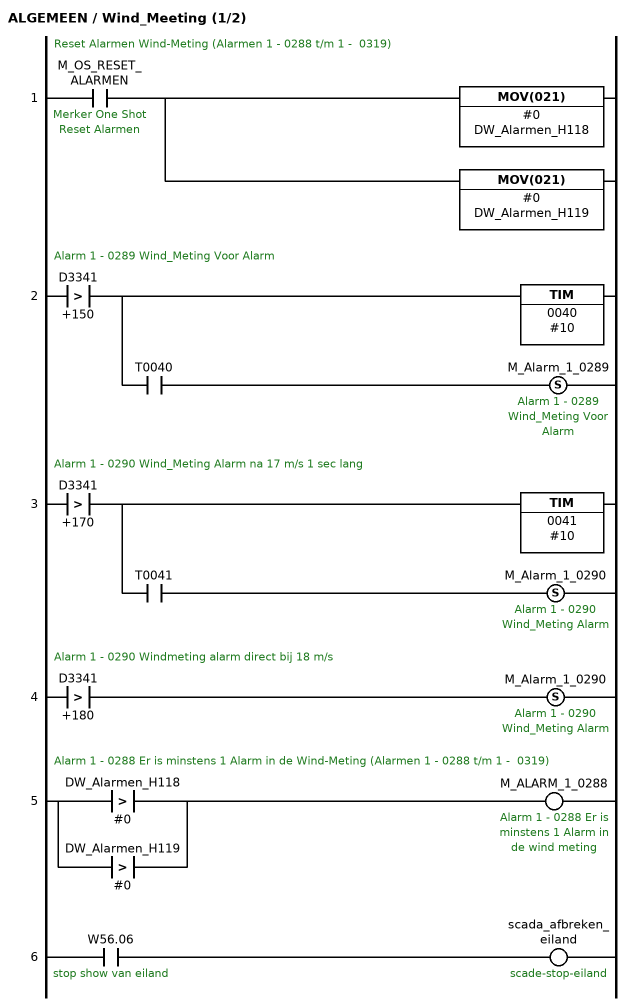
; [picture p72: ALGEMEEN / Wind_Meeting, rungs 1-6]
; rung 1: Reset Alarmen Wind-Meting (Alarmen 1 - 0288 t/m 1 -  0319)
LD M_OS_RESET_ALARMEN  ; Merker One Shot Reset Alarmen
MOV(021) #0 DW_Alarmen_H118
MOV(021) #0 DW_Alarmen_H119
; rung 2: Alarm 1 - 0289 Wind_Meting Voor Alarm
LD>S(322) D3341 +150
TIM 0040 #10
AND T0040
SET M_Alarm_1_0289  ; Alarm 1 - 0289 Wind_Meting Voor Alarm
; rung 3: Alarm 1 - 0290 Wind_Meting Alarm na 17 m/s 1 sec lang
LD>S(322) D3341 +170
TIM 0041 #10
AND T0041
SET M_Alarm_1_0290  ; Alarm 1 - 0290 Wind_Meting Alarm
; rung 4: Alarm 1 - 0290 Windmeting alarm direct bij 18 m/s
LD>S(322) D3341 +180
SET M_Alarm_1_0290  ; Alarm 1 - 0290 Wind_Meting Alarm
; rung 5: Alarm 1 - 0288 Er is minstens 1 Alarm in de Wind-Meting (Alarmen 1 - 0288 t/m 1 -  0319)
LD>(320) DW_Alarmen_H118 #0
OR>(320) DW_Alarmen_H119 #0
OUT M_ALARM_1_0288  ; Alarm 1 - 0288 Er is minstens 1 Alarm in de wind meting
; rung 6
LD W56.06  ; stop show van eiland
OUT scada_afbreken_eiland  ; scade-stop-eiland

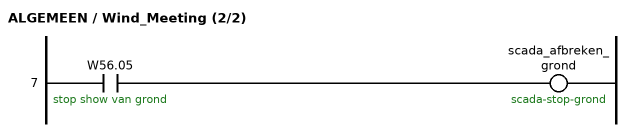
; rung 7
LD W56.05  ; stop show van grond
OUT scada_afbreken_grond  ; scada-stop-grond

### Section Alarm_Handler

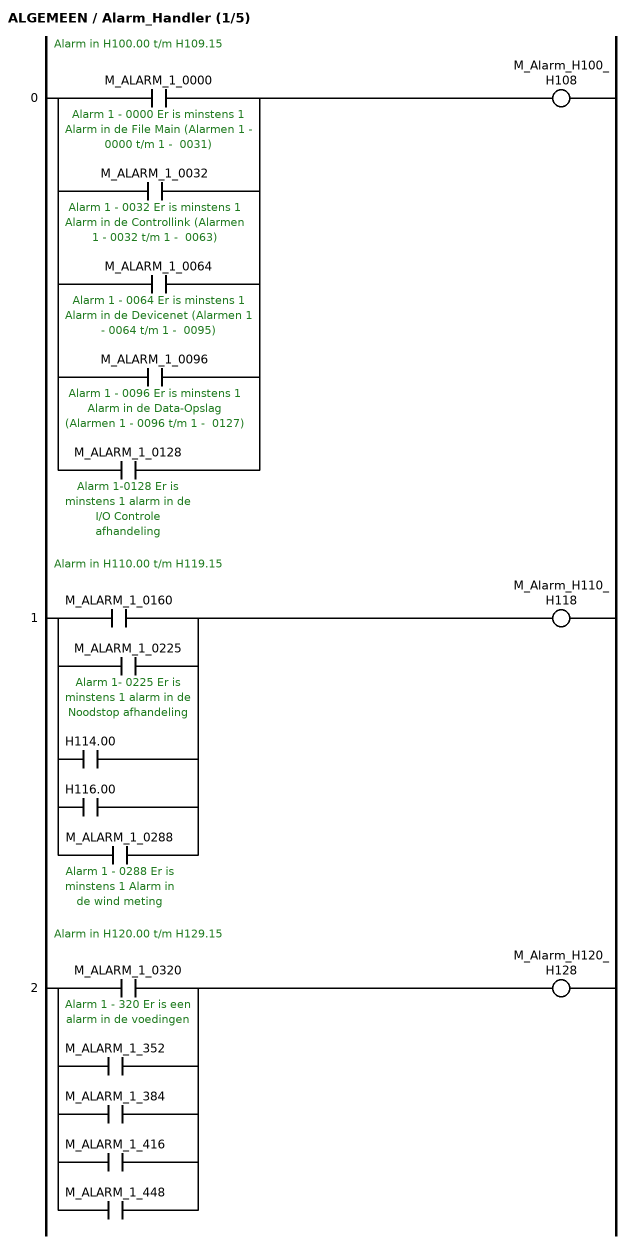
; rung 0: Alarm in H100.00 t/m H109.15
LD M_ALARM_1_0000  ; Alarm 1 - 0000 Er is minstens 1 Alarm in de File Main (Alarmen 1 - 0000 t/m 1 -  0031)
OR M_ALARM_1_0032  ; Alarm 1 - 0032 Er is minstens 1 Alarm in de Controllink (Alarmen 1 - 0032 t/m 1 -  0063)
OR M_ALARM_1_0064  ; Alarm 1 - 0064 Er is minstens 1 Alarm in de Devicenet (Alarmen 1 - 0064 t/m 1 -  0095)
OR M_ALARM_1_0096  ; Alarm 1 - 0096 Er is minstens 1 Alarm in de Data-Opslag (Alarmen 1 - 0096 t/m 1 -  0127)
OR M_ALARM_1_0128  ; Alarm 1-0128 Er is minstens 1 alarm in de I/O Controle afhandeling
OUT M_Alarm_H100_H108
; rung 1: Alarm in H110.00 t/m H119.15
LD M_ALARM_1_0160
OR M_ALARM_1_0225  ; Alarm 1- 0225 Er is minstens 1 alarm in de Noodstop afhandeling
OR H114.00
OR H116.00
OR M_ALARM_1_0288  ; Alarm 1 - 0288 Er is minstens 1 Alarm in de wind meting
OUT M_Alarm_H110_H118
; rung 2: Alarm in H120.00 t/m H129.15
LD M_ALARM_1_0320  ; Alarm 1 - 320 Er is een alarm in de voedingen
OR M_ALARM_1_352
OR M_ALARM_1_384
OR M_ALARM_1_416
OR M_ALARM_1_448
OUT M_Alarm_H120_H128

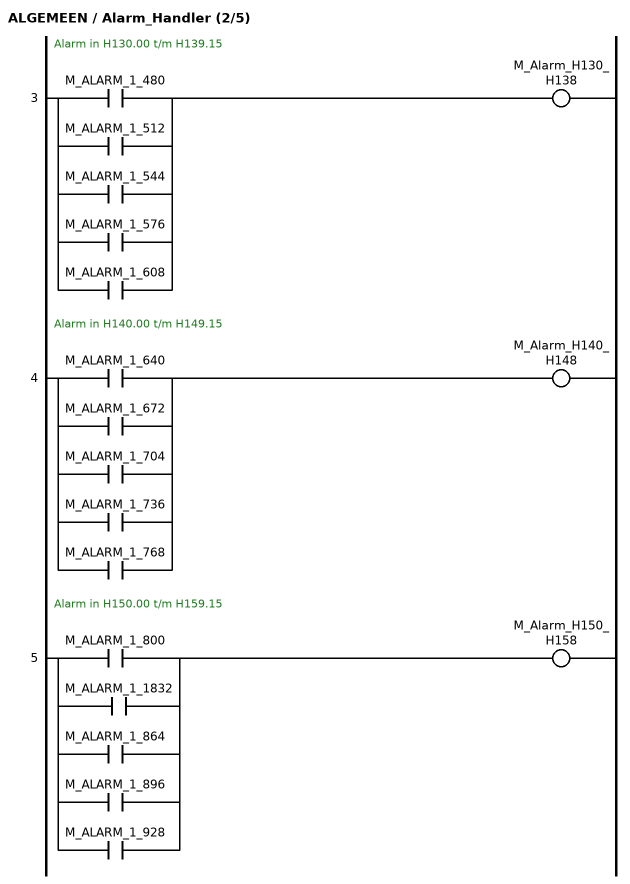
; rung 3: Alarm in H130.00 t/m H139.15
LD M_ALARM_1_480
OR M_ALARM_1_512
OR M_ALARM_1_544
OR M_ALARM_1_576
OR M_ALARM_1_608
OUT M_Alarm_H130_H138
; rung 4: Alarm in H140.00 t/m H149.15
LD M_ALARM_1_640
OR M_ALARM_1_672
OR M_ALARM_1_704
OR M_ALARM_1_736
OR M_ALARM_1_768
OUT M_Alarm_H140_H148
; rung 5: Alarm in H150.00 t/m H159.15
LD M_ALARM_1_800
OR M_ALARM_1_1832
OR M_ALARM_1_864
OR M_ALARM_1_896
OR M_ALARM_1_928
OUT M_Alarm_H150_H158

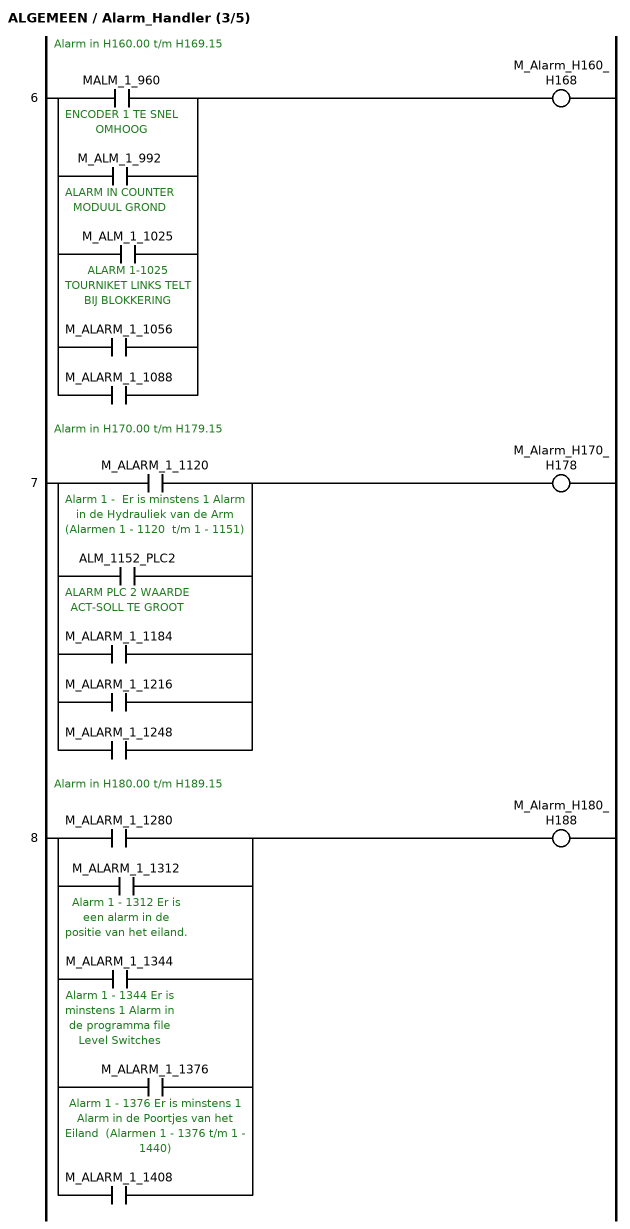
; rung 6: Alarm in H160.00 t/m H169.15
LD MALM_1_960  ; ENCODER 1 TE SNEL OMHOOG
OR M_ALM_1_992  ; ALARM IN COUNTER MODUUL GROND
OR M_ALM_1_1025  ; ALARM 1-1025 TOURNIKET LINKS TELT BIJ BLOKKERING
OR M_ALARM_1_1056
OR M_ALARM_1_1088
OUT M_Alarm_H160_H168
; rung 7: Alarm in H170.00 t/m H179.15
LD M_ALARM_1_1120  ; Alarm 1 -  Er is minstens 1 Alarm in de Hydrauliek van de Arm  (Alarmen 1 - 1120  t/m 1 - 1151)
OR ALM_1152_PLC2  ; ALARM PLC 2 WAARDE ACT-SOLL TE GROOT
OR M_ALARM_1_1184
OR M_ALARM_1_1216
OR M_ALARM_1_1248
OUT M_Alarm_H170_H178
; rung 8: Alarm in H180.00 t/m H189.15
LD M_ALARM_1_1280
OR M_ALARM_1_1312  ; Alarm 1 - 1312 Er is een alarm in de positie van het eiland.
OR M_ALARM_1_1344  ; Alarm 1 - 1344 Er is minstens 1 Alarm in de programma file Level Switches
OR M_ALARM_1_1376  ; Alarm 1 - 1376 Er is minstens 1 Alarm in de Poortjes van het Eiland  (Alarmen 1 - 1376 t/m 1 - 1440)
OR M_ALARM_1_1408
OUT M_Alarm_H180_H188

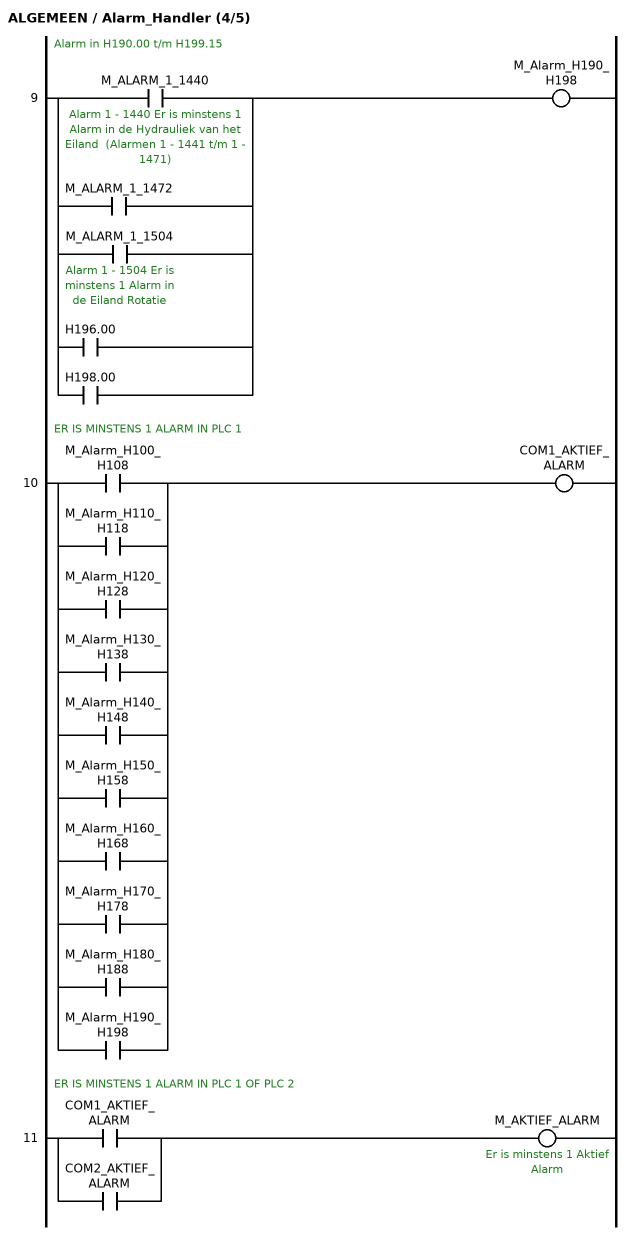
; rung 9: Alarm in H190.00 t/m H199.15
LD M_ALARM_1_1440  ; Alarm 1 - 1440 Er is minstens 1 Alarm in de Hydrauliek van het Eiland  (Alarmen 1 - 1441 t/m 1 - 1471)
OR M_ALARM_1_1472
OR M_ALARM_1_1504  ; Alarm 1 - 1504 Er is minstens 1 Alarm in de Eiland Rotatie
OR H196.00
OR H198.00
OUT M_Alarm_H190_H198
; rung 10: ER IS MINSTENS 1 ALARM IN PLC 1
LD M_Alarm_H100_H108
OR M_Alarm_H110_H118
OR M_Alarm_H120_H128
OR M_Alarm_H130_H138
OR M_Alarm_H140_H148
OR M_Alarm_H150_H158
OR M_Alarm_H160_H168
OR M_Alarm_H170_H178
OR M_Alarm_H180_H188
OR M_Alarm_H190_H198
OUT COM1_AKTIEF_ALARM
; rung 11: ER IS MINSTENS 1 ALARM IN PLC 1 OF PLC 2
LD COM1_AKTIEF_ALARM
OR COM2_AKTIEF_ALARM
OUT M_AKTIEF_ALARM  ; Er is minstens 1 Aktief Alarm

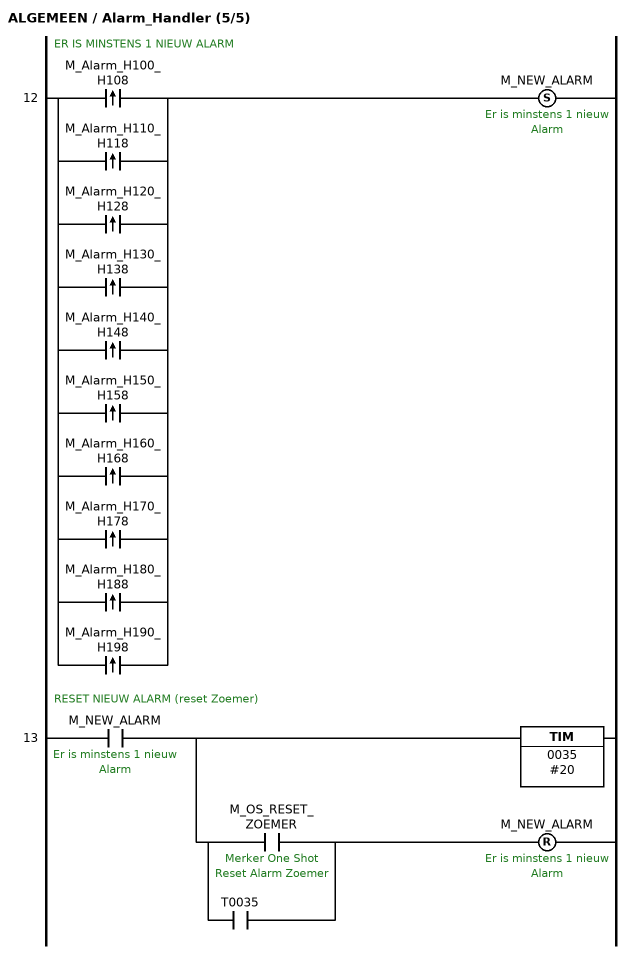
; rung 12: ER IS MINSTENS 1 NIEUW ALARM
@LD M_Alarm_H100_H108
@OR M_Alarm_H110_H118
@OR M_Alarm_H120_H128
@OR M_Alarm_H130_H138
@OR M_Alarm_H140_H148
@OR M_Alarm_H150_H158
@OR M_Alarm_H160_H168
@OR M_Alarm_H170_H178
@OR M_Alarm_H180_H188
@OR M_Alarm_H190_H198
SET M_NEW_ALARM  ; Er is minstens 1 nieuw Alarm
; rung 13: RESET NIEUW ALARM (reset Zoemer)
LD M_NEW_ALARM  ; Er is minstens 1 nieuw Alarm
TIM 0035 #20
LD M_OS_RESET_ZOEMER  ; Merker One Shot Reset Alarm Zoemer
OR T0035
ANDLD
RSET M_NEW_ALARM  ; Er is minstens 1 nieuw Alarm

### Section Einde_Algemeen
; rung 0
END(001)

## Program BEDIENING_SIGNAAL (cyclic task 1)
Local symbols
M_Hydrauliek_x_tijd_aan W56.03 BOOL  ; Hydrauliek x tijd laten door lopen nadat mode is veranderd

### Section Bediening_Scada

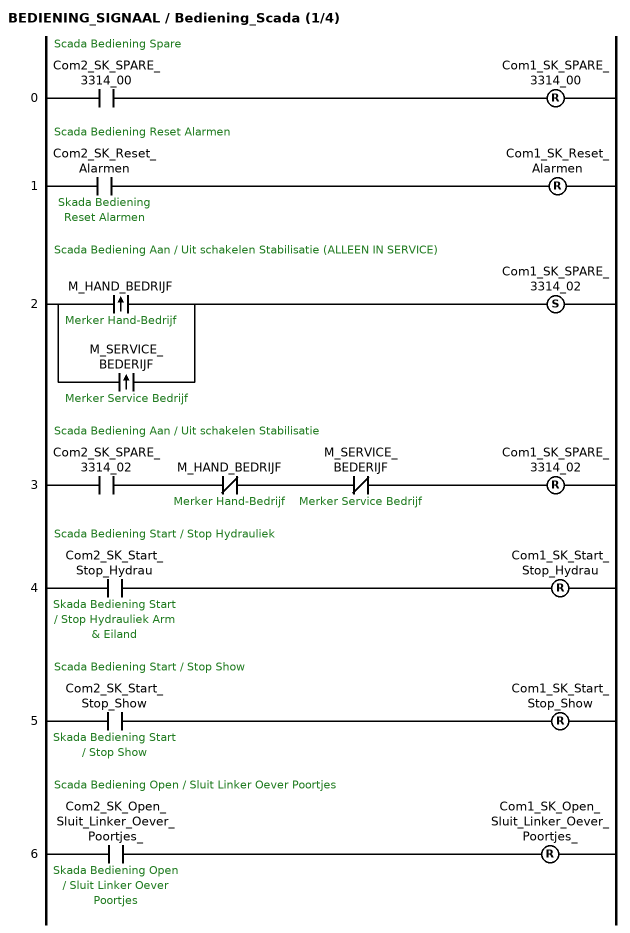
; rung 0: Scada Bediening Spare
LD Com2_SK_SPARE_3314_00
RSET Com1_SK_SPARE_3314_00
; rung 1: Scada Bediening Reset Alarmen
LD Com2_SK_Reset_Alarmen  ; Skada Bediening Reset Alarmen
RSET Com1_SK_Reset_Alarmen
; rung 2: Scada Bediening Aan / Uit schakelen Stabilisatie (ALLEEN IN SERVICE)
@LD M_HAND_BEDRIJF  ; Merker Hand-Bedrijf
@OR M_SERVICE_BEDERIJF  ; Merker Service Bedrijf
SET Com1_SK_SPARE_3314_02
; rung 3: Scada Bediening Aan / Uit schakelen Stabilisatie
LD Com2_SK_SPARE_3314_02
ANDNOT M_HAND_BEDRIJF  ; Merker Hand-Bedrijf
ANDNOT M_SERVICE_BEDERIJF  ; Merker Service Bedrijf
RSET Com1_SK_SPARE_3314_02
; rung 4: Scada Bediening Start / Stop Hydrauliek
LD Com2_SK_Start_Stop_Hydrau  ; Skada Bediening Start / Stop Hydrauliek Arm & Eiland
RSET Com1_SK_Start_Stop_Hydrau
; rung 5: Scada Bediening Start / Stop Show
LD Com2_SK_Start_Stop_Show  ; Skada Bediening Start / Stop Show
RSET Com1_SK_Start_Stop_Show
; rung 6: Scada Bediening Open / Sluit Linker Oever Poortjes
LD Com2_SK_Open_Sluit_Linker_Oever_Poortjes_  ; Skada Bediening Open / Sluit Linker Oever Poortjes
RSET Com1_SK_Open_Sluit_Linker_Oever_Poortjes_

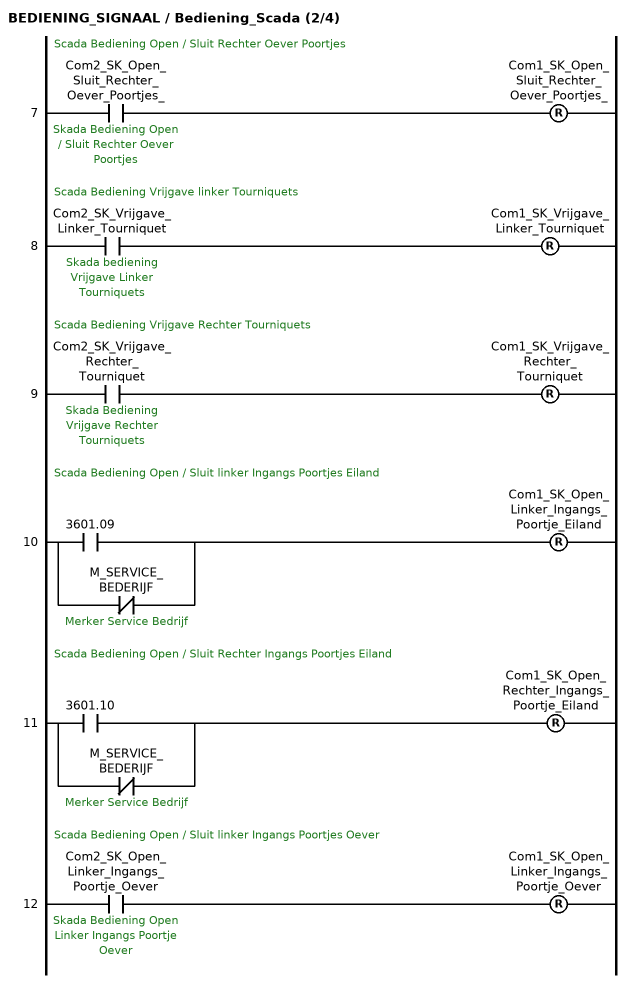
; rung 7: Scada Bediening Open / Sluit Rechter Oever Poortjes
LD Com2_SK_Open_Sluit_Rechter_Oever_Poortjes_  ; Skada Bediening Open / Sluit Rechter Oever Poortjes
RSET Com1_SK_Open_Sluit_Rechter_Oever_Poortjes_
; rung 8: Scada Bediening Vrijgave linker Tourniquets
LD Com2_SK_Vrijgave_Linker_Tourniquet  ; Skada bediening Vrijgave Linker Tourniquets
RSET Com1_SK_Vrijgave_Linker_Tourniquet
; rung 9: Scada Bediening Vrijgave Rechter Tourniquets
LD Com2_SK_Vrijgave_Rechter_Tourniquet  ; Skada Bediening Vrijgave Rechter Tourniquets
RSET Com1_SK_Vrijgave_Rechter_Tourniquet
; rung 10: Scada Bediening Open / Sluit linker Ingangs Poortjes Eiland
LD 3601.09
ORNOT M_SERVICE_BEDERIJF  ; Merker Service Bedrijf
RSET Com1_SK_Open_Linker_Ingangs_Poortje_Eiland
; rung 11: Scada Bediening Open / Sluit Rechter Ingangs Poortjes Eiland
LD 3601.10
ORNOT M_SERVICE_BEDERIJF  ; Merker Service Bedrijf
RSET Com1_SK_Open_Rechter_Ingangs_Poortje_Eiland
; rung 12: Scada Bediening Open / Sluit linker Ingangs Poortjes Oever
LD Com2_SK_Open_Linker_Ingangs_Poortje_Oever  ; Skada Bediening Open Linker Ingangs Poortje Oever
RSET Com1_SK_Open_Linker_Ingangs_Poortje_Oever

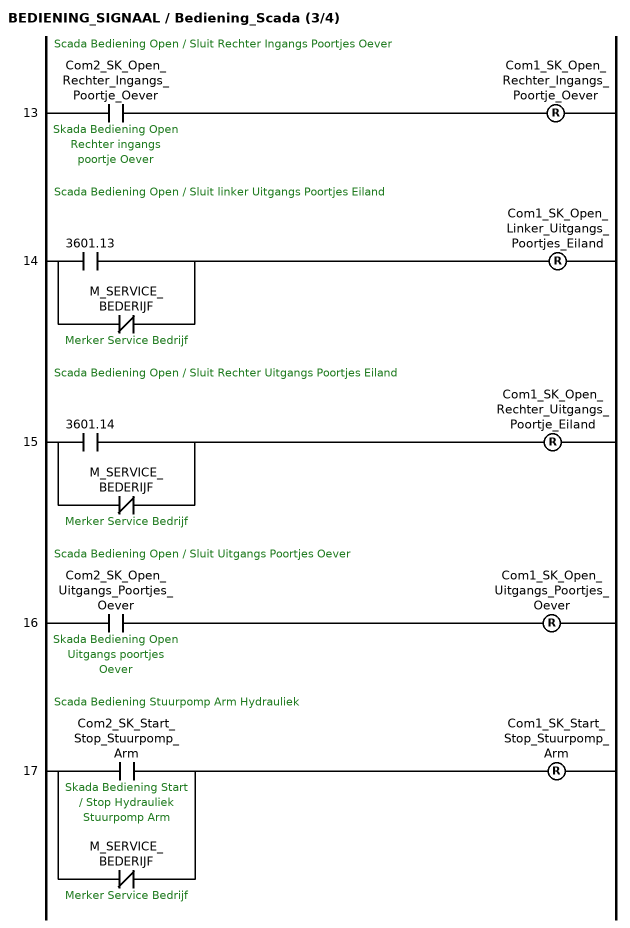
; rung 13: Scada Bediening Open / Sluit Rechter Ingangs Poortjes Oever
LD Com2_SK_Open_Rechter_Ingangs_Poortje_Oever  ; Skada Bediening Open Rechter ingangs poortje Oever
RSET Com1_SK_Open_Rechter_Ingangs_Poortje_Oever
; rung 14: Scada Bediening Open / Sluit linker Uitgangs Poortjes Eiland
LD 3601.13
ORNOT M_SERVICE_BEDERIJF  ; Merker Service Bedrijf
RSET Com1_SK_Open_Linker_Uitgangs_Poortjes_Eiland
; rung 15: Scada Bediening Open / Sluit Rechter Uitgangs Poortjes Eiland
LD 3601.14
ORNOT M_SERVICE_BEDERIJF  ; Merker Service Bedrijf
RSET Com1_SK_Open_Rechter_Uitgangs_Poortje_Eiland
; rung 16: Scada Bediening Open / Sluit Uitgangs Poortjes Oever
LD Com2_SK_Open_Uitgangs_Poortjes_Oever  ; Skada Bediening Open Uitgangs poortjes Oever
RSET Com1_SK_Open_Uitgangs_Poortjes_Oever
; rung 17: Scada Bediening Stuurpomp Arm Hydrauliek
LD Com2_SK_Start_Stop_Stuurpomp_Arm  ; Skada Bediening Start / Stop Hydrauliek Stuurpomp Arm
ORNOT M_SERVICE_BEDERIJF  ; Merker Service Bedrijf
RSET Com1_SK_Start_Stop_Stuurpomp_Arm

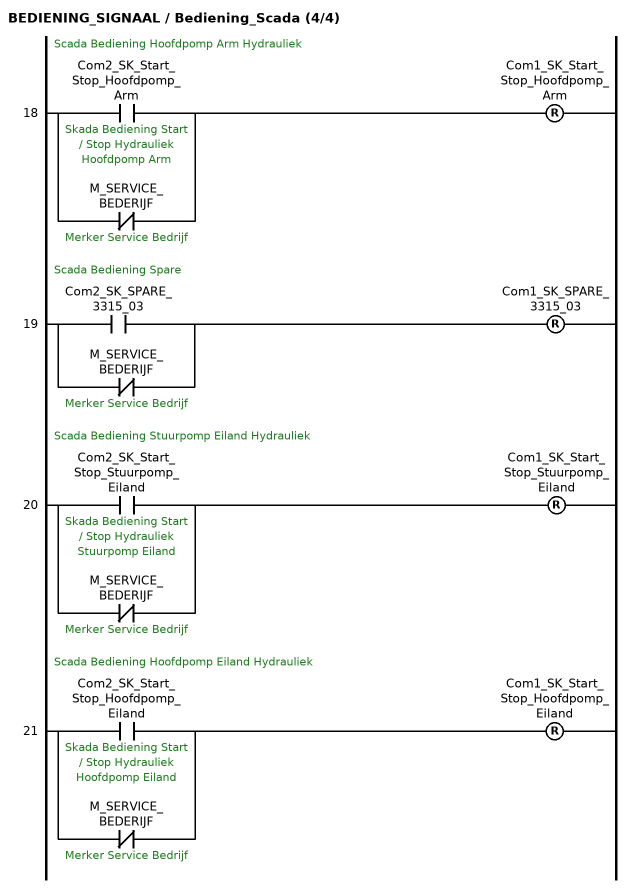
; rung 18: Scada Bediening Hoofdpomp Arm Hydrauliek
LD Com2_SK_Start_Stop_Hoofdpomp_Arm  ; Skada Bediening Start / Stop Hydrauliek Hoofdpomp Arm
ORNOT M_SERVICE_BEDERIJF  ; Merker Service Bedrijf
RSET Com1_SK_Start_Stop_Hoofdpomp_Arm
; rung 19: Scada Bediening Spare
LD Com2_SK_SPARE_3315_03
ORNOT M_SERVICE_BEDERIJF  ; Merker Service Bedrijf
RSET Com1_SK_SPARE_3315_03
; rung 20: Scada Bediening Stuurpomp Eiland Hydrauliek
LD Com2_SK_Start_Stop_Stuurpomp_Eiland  ; Skada Bediening Start / Stop Hydrauliek Stuurpomp Eiland
ORNOT M_SERVICE_BEDERIJF  ; Merker Service Bedrijf
RSET Com1_SK_Start_Stop_Stuurpomp_Eiland
; rung 21: Scada Bediening Hoofdpomp Eiland Hydrauliek
LD Com2_SK_Start_Stop_Hoofdpomp_Eiland  ; Skada Bediening Start / Stop Hydrauliek Hoofdpomp Eiland
ORNOT M_SERVICE_BEDERIJF  ; Merker Service Bedrijf
RSET Com1_SK_Start_Stop_Hoofdpomp_Eiland

### Section Signalering_Scada

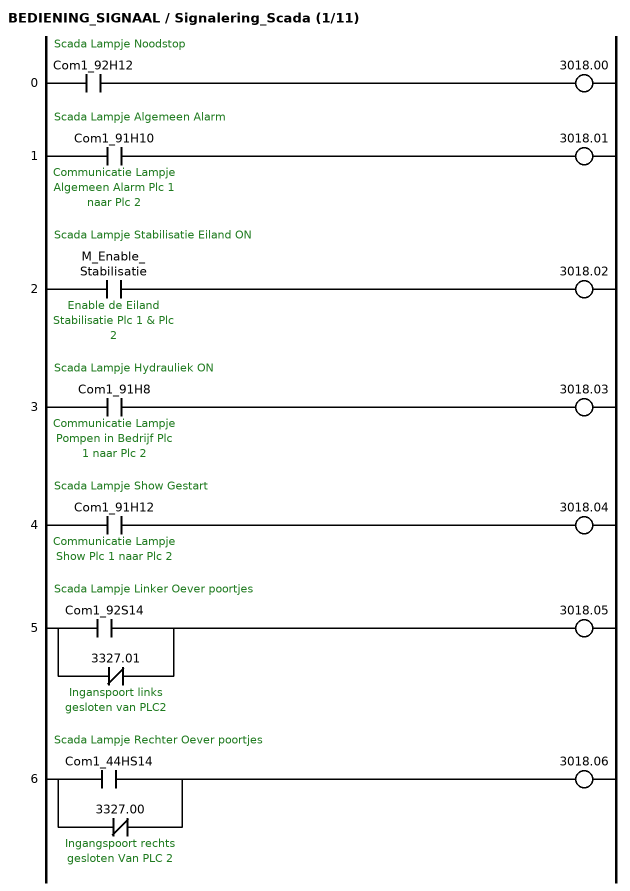
; rung 0: Scada Lampje Noodstop
LD Com1_92H12
OUT 3018.00
; rung 1: Scada Lampje Algemeen Alarm
LD Com1_91H10  ; Communicatie Lampje Algemeen Alarm Plc 1 naar Plc 2
OUT 3018.01
; rung 2: Scada Lampje Stabilisatie Eiland ON
LD M_Enable_Stabilisatie  ; Enable de Eiland Stabilisatie Plc 1 & Plc 2
OUT 3018.02
; rung 3: Scada Lampje Hydrauliek ON
LD Com1_91H8  ; Communicatie Lampje Pompen in Bedrijf Plc 1 naar Plc 2
OUT 3018.03
; rung 4: Scada Lampje Show Gestart
LD Com1_91H12  ; Communicatie Lampje Show Plc 1 naar Plc 2
OUT 3018.04
; rung 5: Scada Lampje Linker Oever poortjes
LD Com1_92S14
ORNOT 3327.01  ; Inganspoort links gesloten van PLC2
OUT 3018.05
; rung 6: Scada Lampje Rechter Oever poortjes
LD Com1_44HS14
ORNOT 3327.00  ; Ingangspoort rechts gesloten Van PLC 2
OUT 3018.06

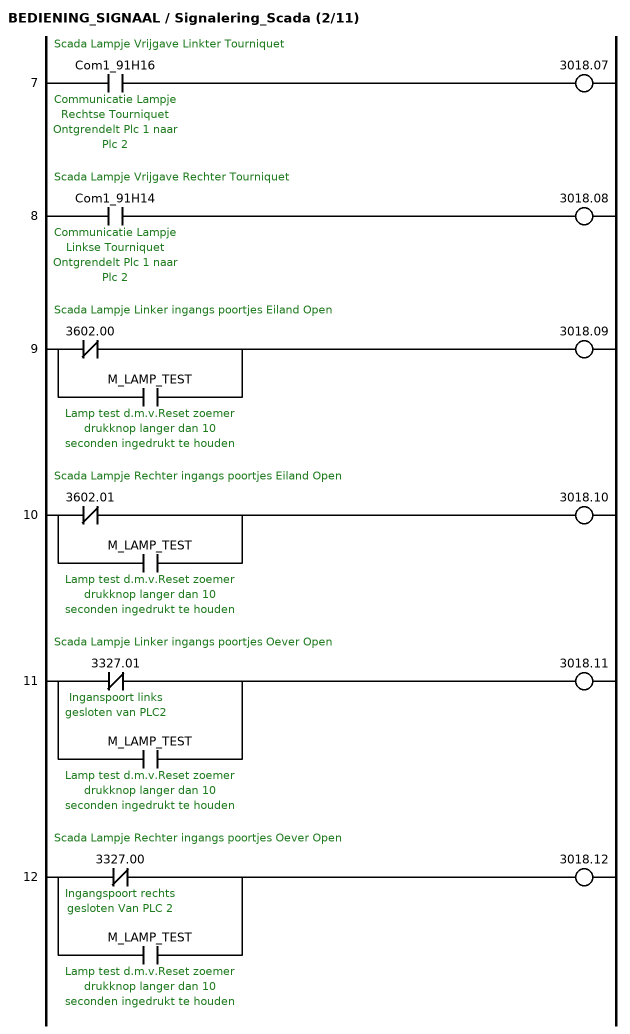
; rung 7: Scada Lampje Vrijgave Linkter Tourniquet
LD Com1_91H16  ; Communicatie Lampje Rechtse Tourniquet Ontgrendelt Plc 1 naar Plc 2
OUT 3018.07
; rung 8: Scada Lampje Vrijgave Rechter Tourniquet
LD Com1_91H14  ; Communicatie Lampje Linkse Tourniquet Ontgrendelt Plc 1 naar Plc 2
OUT 3018.08
; rung 9: Scada Lampje Linker ingangs poortjes Eiland Open
LDNOT 3602.00
OR M_LAMP_TEST  ; Lamp test d.m.v.Reset zoemer drukknop langer dan 10 seconden ingedrukt te houden
OUT 3018.09
; rung 10: Scada Lampje Rechter ingangs poortjes Eiland Open
LDNOT 3602.01
OR M_LAMP_TEST  ; Lamp test d.m.v.Reset zoemer drukknop langer dan 10 seconden ingedrukt te houden
OUT 3018.10
; rung 11: Scada Lampje Linker ingangs poortjes Oever Open
LDNOT 3327.01  ; Inganspoort links gesloten van PLC2
OR M_LAMP_TEST  ; Lamp test d.m.v.Reset zoemer drukknop langer dan 10 seconden ingedrukt te houden
OUT 3018.11
; rung 12: Scada Lampje Rechter ingangs poortjes Oever Open
LDNOT 3327.00  ; Ingangspoort rechts gesloten Van PLC 2
OR M_LAMP_TEST  ; Lamp test d.m.v.Reset zoemer drukknop langer dan 10 seconden ingedrukt te houden
OUT 3018.12

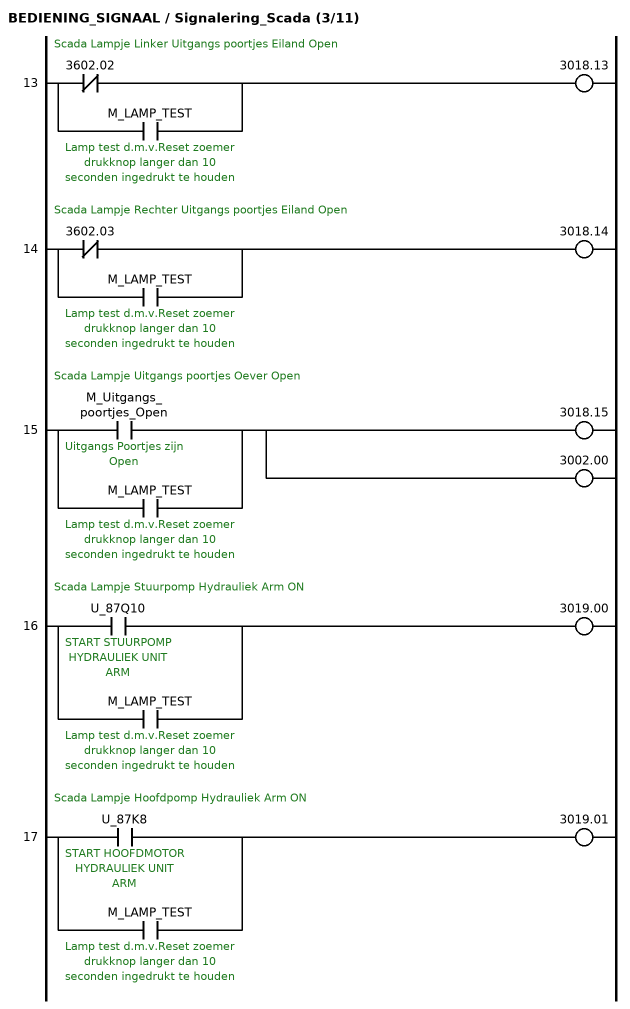
; rung 13: Scada Lampje Linker Uitgangs poortjes Eiland Open
LDNOT 3602.02
OR M_LAMP_TEST  ; Lamp test d.m.v.Reset zoemer drukknop langer dan 10 seconden ingedrukt te houden
OUT 3018.13
; rung 14: Scada Lampje Rechter Uitgangs poortjes Eiland Open
LDNOT 3602.03
OR M_LAMP_TEST  ; Lamp test d.m.v.Reset zoemer drukknop langer dan 10 seconden ingedrukt te houden
OUT 3018.14
; rung 15: Scada Lampje Uitgangs poortjes Oever Open
LD M_Uitgangs_poortjes_Open  ; Uitgangs Poortjes zijn Open
OR M_LAMP_TEST  ; Lamp test d.m.v.Reset zoemer drukknop langer dan 10 seconden ingedrukt te houden
OUT 3018.15
OUT 3002.00
; rung 16: Scada Lampje Stuurpomp Hydrauliek Arm ON
LD U_87Q10  ; START STUURPOMP HYDRAULIEK UNIT ARM
OR M_LAMP_TEST  ; Lamp test d.m.v.Reset zoemer drukknop langer dan 10 seconden ingedrukt te houden
OUT 3019.00
; rung 17: Scada Lampje Hoofdpomp Hydrauliek Arm ON
LD U_87K8  ; START HOOFDMOTOR HYDRAULIEK UNIT ARM
OR M_LAMP_TEST  ; Lamp test d.m.v.Reset zoemer drukknop langer dan 10 seconden ingedrukt te houden
OUT 3019.01

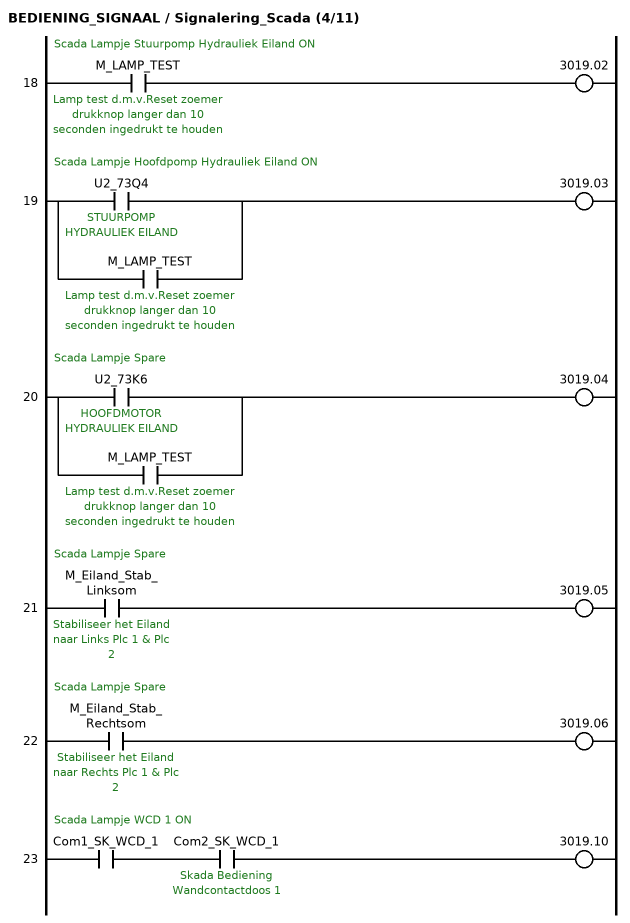
; rung 18: Scada Lampje Stuurpomp Hydrauliek Eiland ON
LD M_LAMP_TEST  ; Lamp test d.m.v.Reset zoemer drukknop langer dan 10 seconden ingedrukt te houden
OUT 3019.02
; rung 19: Scada Lampje Hoofdpomp Hydrauliek Eiland ON
LD U2_73Q4  ; STUURPOMP HYDRAULIEK EILAND
OR M_LAMP_TEST  ; Lamp test d.m.v.Reset zoemer drukknop langer dan 10 seconden ingedrukt te houden
OUT 3019.03
; rung 20: Scada Lampje Spare
LD U2_73K6  ; HOOFDMOTOR HYDRAULIEK EILAND
OR M_LAMP_TEST  ; Lamp test d.m.v.Reset zoemer drukknop langer dan 10 seconden ingedrukt te houden
OUT 3019.04
; rung 21: Scada Lampje Spare
LD M_Eiland_Stab_Linksom  ; Stabiliseer het Eiland naar Links Plc 1 & Plc 2
OUT 3019.05
; rung 22: Scada Lampje Spare
LD M_Eiland_Stab_Rechtsom  ; Stabiliseer het Eiland naar Rechts Plc 1 & Plc 2
OUT 3019.06
; rung 23: Scada Lampje WCD 1 ON
LD Com1_SK_WCD_1
AND Com2_SK_WCD_1  ; Skada Bediening Wandcontactdoos 1
OUT 3019.10

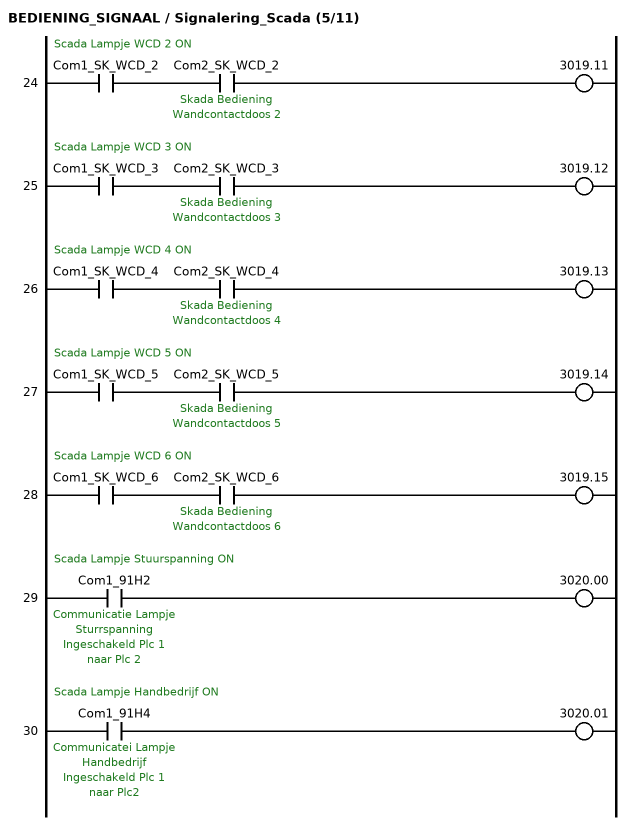
; rung 24: Scada Lampje WCD 2 ON
LD Com1_SK_WCD_2
AND Com2_SK_WCD_2  ; Skada Bediening Wandcontactdoos 2
OUT 3019.11
; rung 25: Scada Lampje WCD 3 ON
LD Com1_SK_WCD_3
AND Com2_SK_WCD_3  ; Skada Bediening Wandcontactdoos 3
OUT 3019.12
; rung 26: Scada Lampje WCD 4 ON
LD Com1_SK_WCD_4
AND Com2_SK_WCD_4  ; Skada Bediening Wandcontactdoos 4
OUT 3019.13
; rung 27: Scada Lampje WCD 5 ON
LD Com1_SK_WCD_5
AND Com2_SK_WCD_5  ; Skada Bediening Wandcontactdoos 5
OUT 3019.14
; rung 28: Scada Lampje WCD 6 ON
LD Com1_SK_WCD_6
AND Com2_SK_WCD_6  ; Skada Bediening Wandcontactdoos 6
OUT 3019.15
; rung 29: Scada Lampje Stuurspanning ON
LD Com1_91H2  ; Communicatie Lampje Sturrspanning Ingeschakeld Plc 1 naar Plc 2
OUT 3020.00
; rung 30: Scada Lampje Handbedrijf ON
LD Com1_91H4  ; Communicatei Lampje Handbedrijf Ingeschakeld Plc 1 naar Plc2
OUT 3020.01

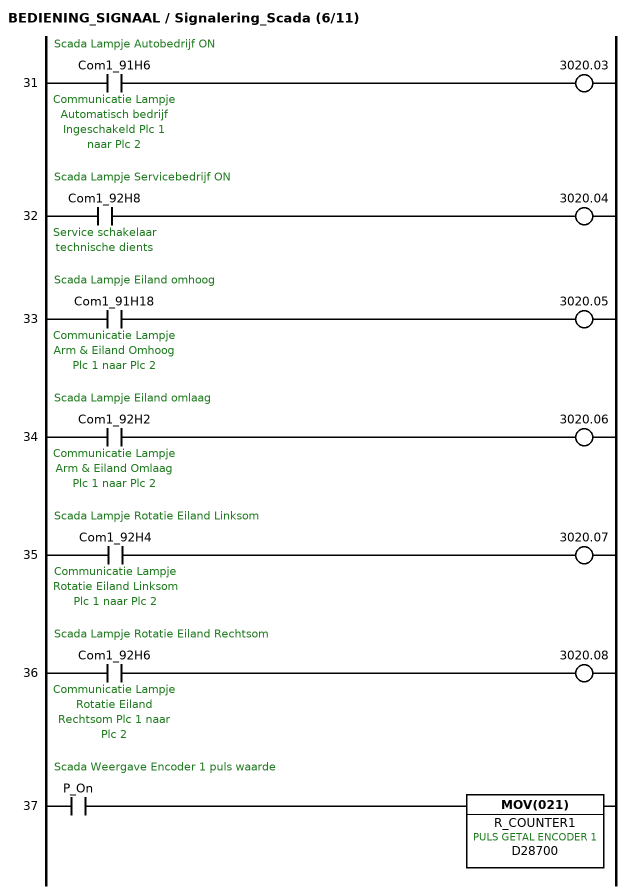
; rung 31: Scada Lampje Autobedrijf ON
LD Com1_91H6  ; Communicatie Lampje Automatisch bedrijf Ingeschakeld Plc 1 naar Plc 2
OUT 3020.03
; rung 32: Scada Lampje Servicebedrijf ON
LD Com1_92H8  ; Service schakelaar technische dients
OUT 3020.04
; rung 33: Scada Lampje Eiland omhoog
LD Com1_91H18  ; Communicatie Lampje Arm & Eiland Omhoog Plc 1 naar Plc 2
OUT 3020.05
; rung 34: Scada Lampje Eiland omlaag
LD Com1_92H2  ; Communicatie Lampje Arm & Eiland Omlaag Plc 1 naar Plc 2
OUT 3020.06
; rung 35: Scada Lampje Rotatie Eiland Linksom
LD Com1_92H4  ; Communicatie Lampje Rotatie Eiland Linksom Plc 1 naar Plc 2
OUT 3020.07
; rung 36: Scada Lampje Rotatie Eiland Rechtsom
LD Com1_92H6  ; Communicatie Lampje Rotatie Eiland Rechtsom Plc 1 naar Plc 2
OUT 3020.08
; rung 37: Scada Weergave Encoder 1 puls waarde
LD P_On
MOV(021) R_COUNTER1 D28700  ; PULS GETAL ENCODER 1

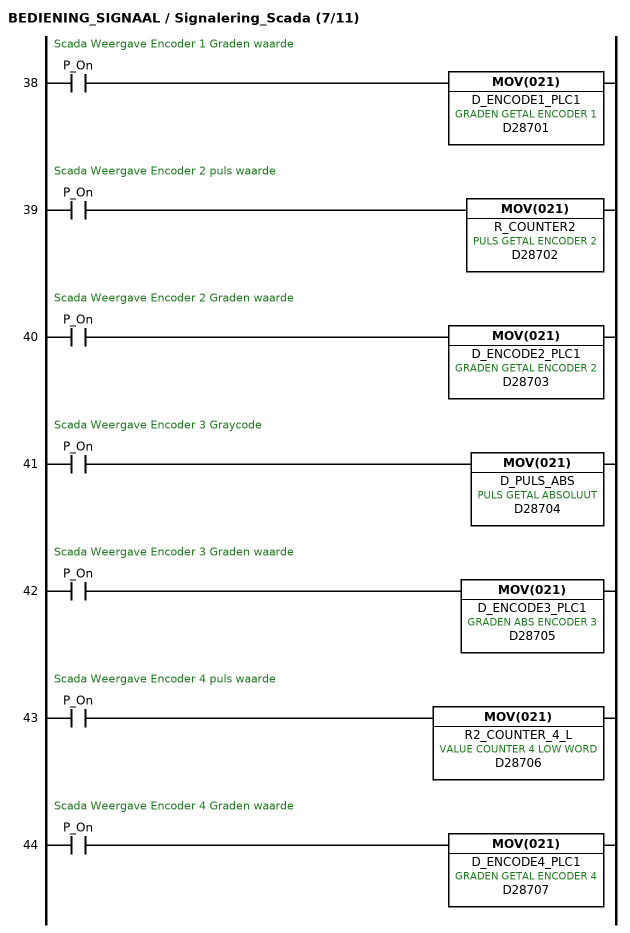
; rung 38: Scada Weergave Encoder 1 Graden waarde
LD P_On
MOV(021) D_ENCODE1_PLC1 D28701  ; GRADEN GETAL ENCODER 1
; rung 39: Scada Weergave Encoder 2 puls waarde
LD P_On
MOV(021) R_COUNTER2 D28702  ; PULS GETAL ENCODER 2
; rung 40: Scada Weergave Encoder 2 Graden waarde
LD P_On
MOV(021) D_ENCODE2_PLC1 D28703  ; GRADEN GETAL ENCODER 2
; rung 41: Scada Weergave Encoder 3 Graycode
LD P_On
MOV(021) D_PULS_ABS D28704  ; PULS GETAL ABSOLUUT
; rung 42: Scada Weergave Encoder 3 Graden waarde
LD P_On
MOV(021) D_ENCODE3_PLC1 D28705  ; GRADEN ABS ENCODER 3
; rung 43: Scada Weergave Encoder 4 puls waarde
LD P_On
MOV(021) R2_COUNTER_4_L D28706  ; VALUE COUNTER 4 LOW WORD
; rung 44: Scada Weergave Encoder 4 Graden waarde
LD P_On
MOV(021) D_ENCODE4_PLC1 D28707  ; GRADEN GETAL ENCODER 4

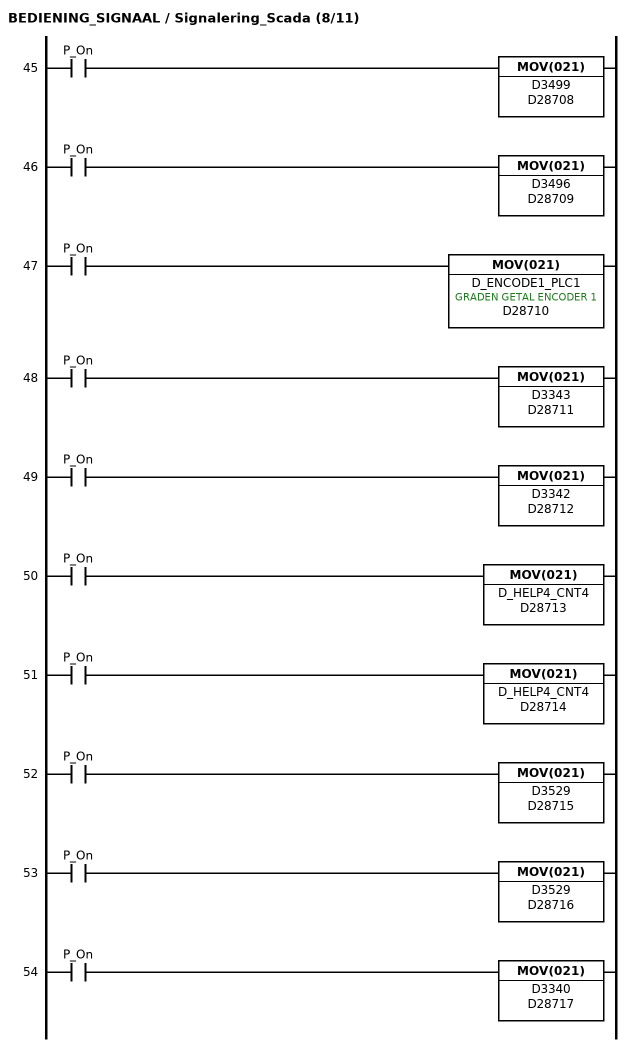
; rung 45
LD P_On
MOV(021) D3499 D28708
; rung 46
LD P_On
MOV(021) D3496 D28709
; rung 47
LD P_On
MOV(021) D_ENCODE1_PLC1 D28710  ; GRADEN GETAL ENCODER 1
; rung 48
LD P_On
MOV(021) D3343 D28711
; rung 49
LD P_On
MOV(021) D3342 D28712
; rung 50
LD P_On
MOV(021) D_HELP4_CNT4 D28713
; rung 51
LD P_On
MOV(021) D_HELP4_CNT4 D28714
; rung 52
LD P_On
MOV(021) D3529 D28715
; rung 53
LD P_On
MOV(021) D3529 D28716
; rung 54
LD P_On
MOV(021) D3340 D28717

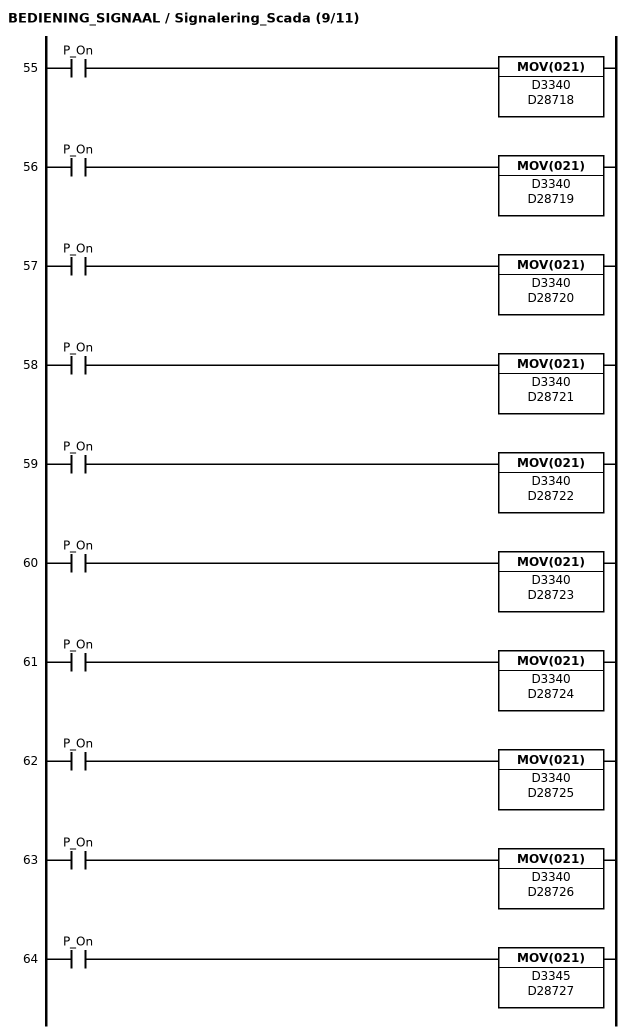
; rung 55
LD P_On
MOV(021) D3340 D28718
; rung 56
LD P_On
MOV(021) D3340 D28719
; rung 57
LD P_On
MOV(021) D3340 D28720
; rung 58
LD P_On
MOV(021) D3340 D28721
; rung 59
LD P_On
MOV(021) D3340 D28722
; rung 60
LD P_On
MOV(021) D3340 D28723
; rung 61
LD P_On
MOV(021) D3340 D28724
; rung 62
LD P_On
MOV(021) D3340 D28725
; rung 63
LD P_On
MOV(021) D3340 D28726
; rung 64
LD P_On
MOV(021) D3345 D28727

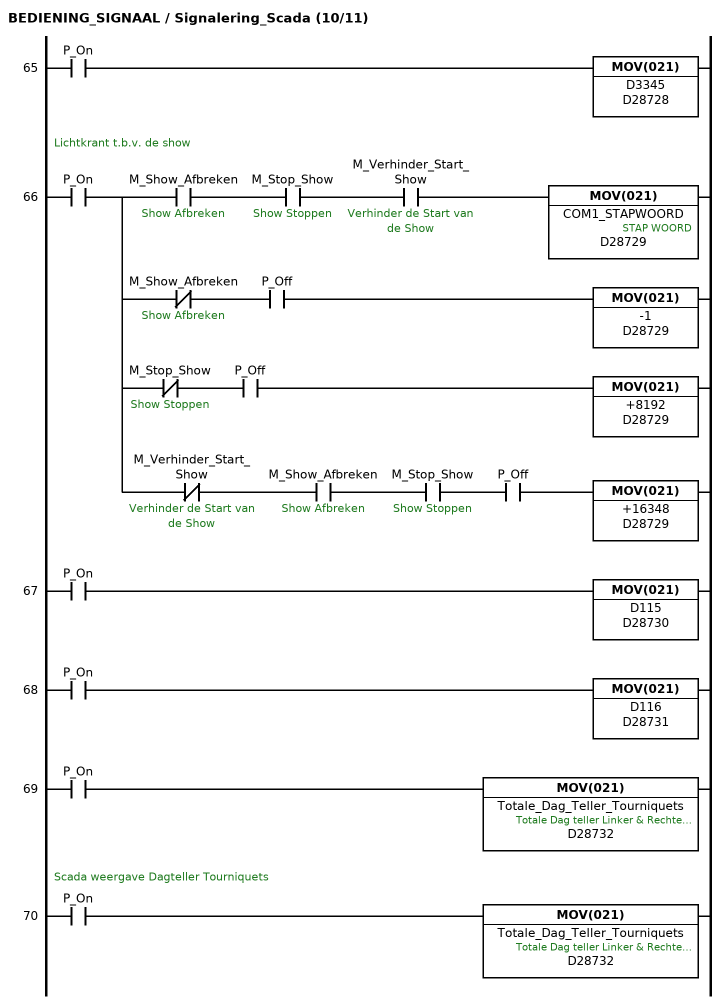
; rung 65
LD P_On
MOV(021) D3345 D28728
; rung 66: Lichtkrant t.b.v. de show
LD P_On
OUT TR0
AND M_Show_Afbreken  ; Show Afbreken
AND M_Stop_Show  ; Show Stoppen
AND M_Verhinder_Start_Show  ; Verhinder de Start van de Show
MOV(021) COM1_STAPWOORD D28729  ; STAP WOORD
LD TR0
ANDNOT M_Show_Afbreken  ; Show Afbreken
AND P_Off
MOV(021) -1 D28729
LD TR0
ANDNOT M_Stop_Show  ; Show Stoppen
AND P_Off
MOV(021) +8192 D28729
LD TR0
ANDNOT M_Verhinder_Start_Show  ; Verhinder de Start van de Show
AND M_Show_Afbreken  ; Show Afbreken
AND M_Stop_Show  ; Show Stoppen
AND P_Off
MOV(021) +16348 D28729
; rung 67
LD P_On
MOV(021) D115 D28730
; rung 68
LD P_On
MOV(021) D116 D28731
; rung 69
LD P_On
MOV(021) Totale_Dag_Teller_Tourniquets D28732  ; Totale Dag teller Linker & Rechter Tournoquets
; rung 70: Scada weergave Dagteller Tourniquets
LD P_On
MOV(021) Totale_Dag_Teller_Tourniquets D28732  ; Totale Dag teller Linker & Rechter Tournoquets

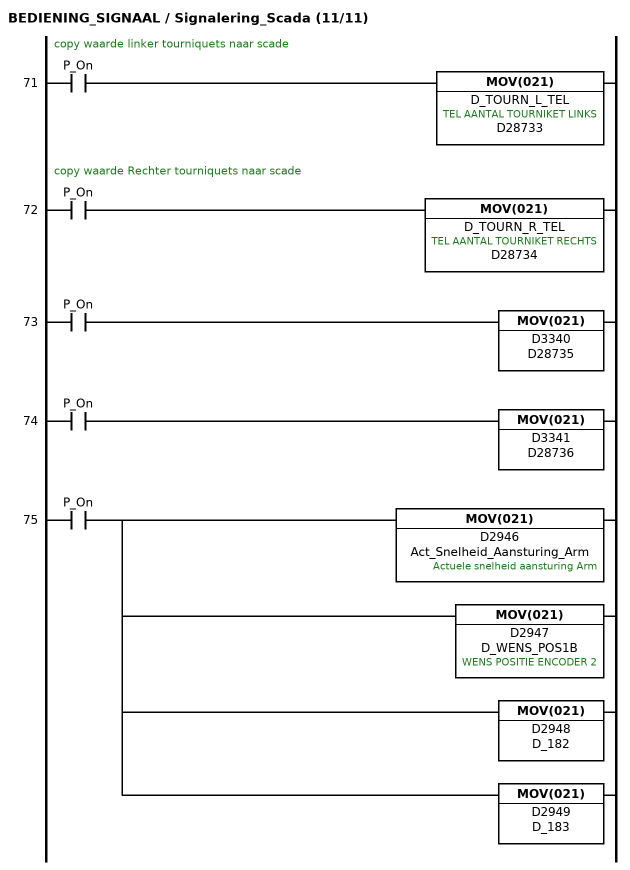
; rung 71: copy waarde linker tourniquets naar scade
LD P_On
MOV(021) D_TOURN_L_TEL D28733  ; TEL AANTAL TOURNIKET LINKS
; rung 72: copy waarde Rechter tourniquets naar scade
LD P_On
MOV(021) D_TOURN_R_TEL D28734  ; TEL AANTAL TOURNIKET RECHTS
; rung 73
LD P_On
MOV(021) D3340 D28735
; rung 74
LD P_On
MOV(021) D3341 D28736
; rung 75
LD P_On
MOV(021) D2946 Act_Snelheid_Aansturing_Arm  ; Actuele snelheid aansturing Arm
MOV(021) D2947 D_WENS_POS1B  ; WENS POSITIE ENCODER 2
MOV(021) D2948 D_182
MOV(021) D2949 D_183

### Section Bediening_Grond

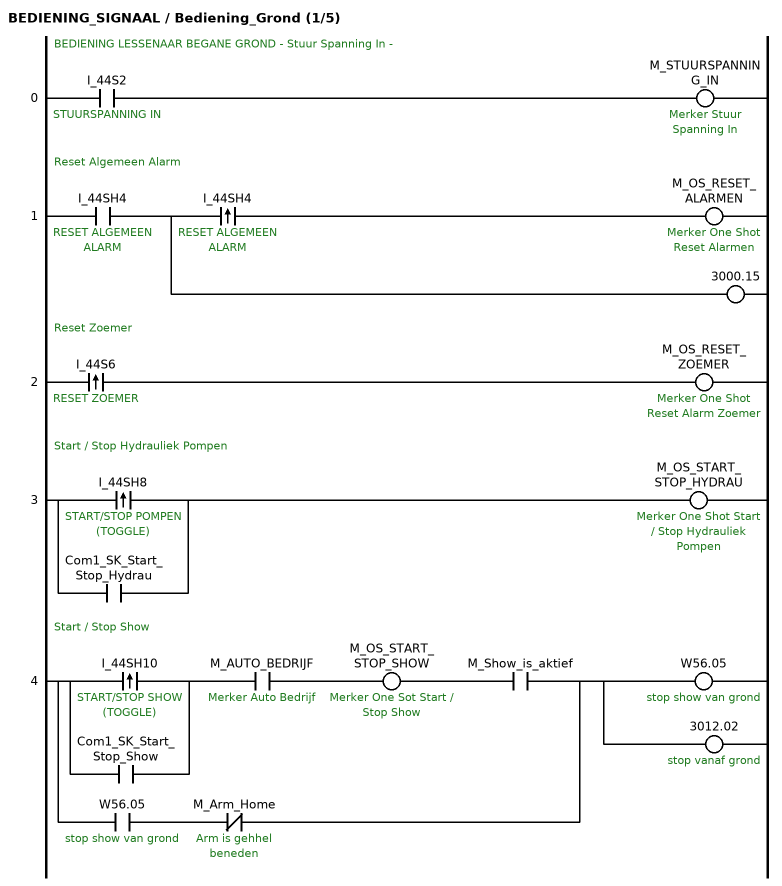
; rung 0: BEDIENING LESSENAAR BEGANE GROND - Stuur Spanning In -
LD I_44S2  ; STUURSPANNING IN
OUT M_STUURSPANNING_IN  ; Merker Stuur Spanning In
; rung 1: Reset Algemeen Alarm
LD I_44SH4  ; RESET ALGEMEEN ALARM
OUT TR0
@AND I_44SH4  ; RESET ALGEMEEN ALARM
OUT M_OS_RESET_ALARMEN  ; Merker One Shot Reset Alarmen
LD TR0
OUT 3000.15
; rung 2: Reset Zoemer
@LD I_44S6  ; RESET ZOEMER
OUT M_OS_RESET_ZOEMER  ; Merker One Shot Reset Alarm Zoemer
; rung 3: Start / Stop Hydrauliek Pompen
@LD I_44SH8  ; START/STOP POMPEN (TOGGLE)
OR Com1_SK_Start_Stop_Hydrau
OUT M_OS_START_STOP_HYDRAU  ; Merker One Shot Start / Stop Hydrauliek Pompen
; rung 4: Start / Stop Show
@LD I_44SH10  ; START/STOP SHOW (TOGGLE)
OR Com1_SK_Start_Stop_Show
AND M_AUTO_BEDRIJF  ; Merker Auto Bedrijf
OUT M_OS_START_STOP_SHOW  ; Merker One Sot Start / Stop Show
AND M_Show_is_aktief
LD W56.05  ; stop show van grond
ANDNOT M_Arm_Home  ; Arm is gehhel beneden
ORLD
OUT W56.05  ; stop show van grond
OUT 3012.02  ; stop vanaf grond

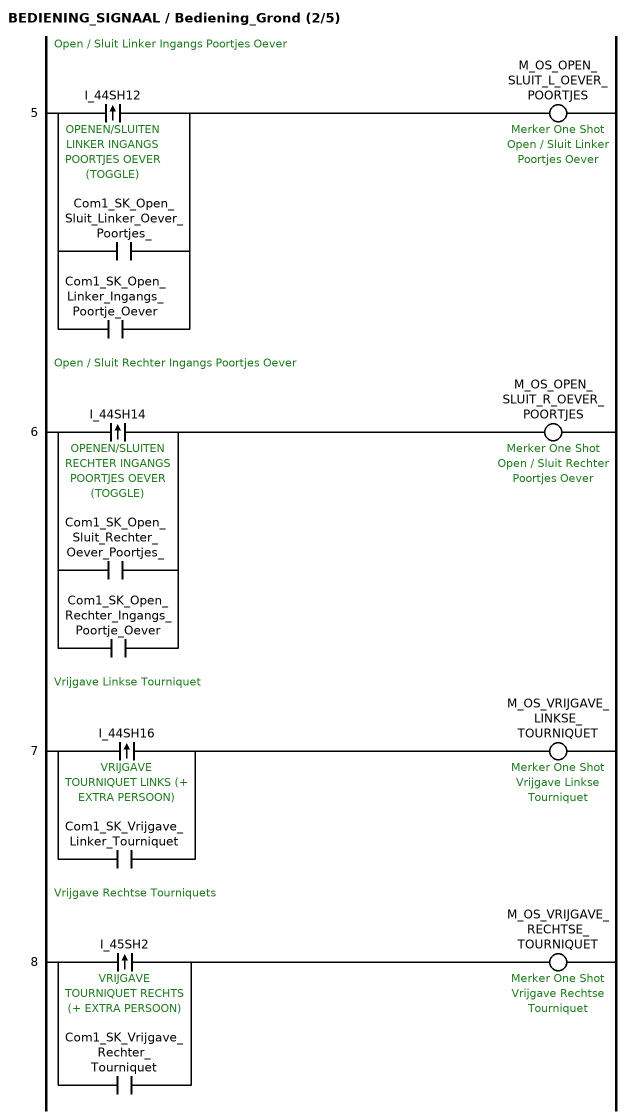
; rung 5: Open / Sluit Linker Ingangs Poortjes Oever
@LD I_44SH12  ; OPENEN/SLUITEN LINKER INGANGS POORTJES OEVER  (TOGGLE)
OR Com1_SK_Open_Sluit_Linker_Oever_Poortjes_
OR Com1_SK_Open_Linker_Ingangs_Poortje_Oever
OUT M_OS_OPEN_SLUIT_L_OEVER_POORTJES  ; Merker One Shot Open / Sluit Linker Poortjes Oever
; rung 6: Open / Sluit Rechter Ingangs Poortjes Oever
@LD I_44SH14  ; OPENEN/SLUITEN RECHTER INGANGS POORTJES OEVER  (TOGGLE)
OR Com1_SK_Open_Sluit_Rechter_Oever_Poortjes_
OR Com1_SK_Open_Rechter_Ingangs_Poortje_Oever
OUT M_OS_OPEN_SLUIT_R_OEVER_POORTJES  ; Merker One Shot Open / Sluit Rechter Poortjes Oever
; rung 7: Vrijgave Linkse Tourniquet
@LD I_44SH16  ; VRIJGAVE TOURNIQUET LINKS (+ EXTRA PERSOON)
OR Com1_SK_Vrijgave_Linker_Tourniquet
OUT M_OS_VRIJGAVE_LINKSE_TOURNIQUET  ; Merker One Shot Vrijgave Linkse Tourniquet
; rung 8: Vrijgave Rechtse Tourniquets
@LD I_45SH2  ; VRIJGAVE TOURNIQUET RECHTS (+ EXTRA PERSOON)
OR Com1_SK_Vrijgave_Rechter_Tourniquet
OUT M_OS_VRIJGAVE_RECHTSE_TOURNIQUET  ; Merker One Shot Vrijgave Rechtse Tourniquet

